TYPE StructuredData EXTENDS TcoCore.TcoStruct :
STRUCT
	_o1 : StructuredObject(THISSTRUCT);
END_STRUCT
END_TYPE

(* stored: Version 1.1.0.1
   DUT StructuredData: Id {b59be22d-326c-052c-2b31-a218d8f837c3} *)
